FUNCTION_BLOCK AnalogOutput EXTENDS BaseIO
VAR_INPUT
	Value: LREAL;
	Override: BOOL;
	OverrideValue: LREAL;
END_VAR
VAR_OUTPUT
	ProcessValue: LREAL;
	ValueOut: LREAL;
END_VAR
VAR
	InitDone: BOOL;
	TempValue: LREAL;
	OutValue: LREAL;
	Override2: BOOL;
	OverrideValue2: LREAL;
END_VAR
VAR PERSISTENT
	SignedWord: BOOL;
	ProcessMin: DINT := 0;
	ProcessMax: DINT := 16#7FFF;
	MinValue: LREAL := 0;
	MaxValue: LREAL := 1;
	SavedOverride: BOOL;
	SavedOverrideValue: LREAL;
	SavedOverride2: BOOL;
	SavedOverrideValue2: LREAL;
END_VAR

SUPER^();
IF NOT InitDone THEN
	InitDone := TRUE;
	OverrideValue := SavedOverrideValue;
	Override := SavedOverride;	
	OverrideValue2 := SavedOverrideValue2;
	Override2 := SavedOverride2;	
END_IF
TempValue := Value;
IF Override2 THEN
	TempValue := OverrideValue2;
END_IF
IF Override THEN
	TempValue := OverrideValue;
END_IF
OutValue := (LimitValue(TempValue, MinValue, MaxValue) - MinValue) / (MaxValue - MinValue) * (ProcessMax - ProcessMin) + ProcessMin;
IF SignedWord THEN
	IF OutValue < 0 THEN
		OutValue := OutValue + 16#10000;
	END_IF
END_IF
ProcessValue := OutValue;
SavedOverride := Override;
SavedOverrideValue := OverrideValue;
SavedOverride2 := Override2;
SavedOverrideValue2 := OverrideValue2;
ValueOut :=TempValue;

METHOD SetOverride2 : BOOL
VAR_INPUT
	OverrideIN: BOOL;
	OverrideValueIN: LREAL;
END_VAR
Override2 := OverrideIN;
OverrideValue2 := OverrideValueIN;
END_METHOD

END_FUNCTION_BLOCK

(* stored: Version 1.1.0.1, ProductVersion 3.1.4024.4
   POU AnalogOutput: Id {a58007a3-0968-41f1-9032-30ac32fdcbac}, SpecialFunc None
   Method SetOverride2: Id {82b71101-8701-497d-9c48-1762b9a0e028} *)
